(* IEC 61131-3 sources: ev-charging-controller/Communication, 3 files *)

(* ---- CanDecodeHelpers.st ---- *)
(* @brief Raw CAN field -> strict enum conversions
 *
 *  Strict enums cannot be assigned from integers, so each 2-bit field
 *  is mapped explicitly. Unknown codes fall back to the safe value.
 *)
FUNCTION F_ToContactorState : E_ContactorState
VAR_INPUT
    raw : BYTE;       (* 2-bit field, already shifted to bits 1:0 *)
END_VAR
    CASE raw OF
        0: F_ToContactorState := E_ContactorState.CTR_OPEN;
        1: F_ToContactorState := E_ContactorState.CTR_CLOSING;
        2: F_ToContactorState := E_ContactorState.CTR_CLOSED;
    ELSE
        F_ToContactorState := E_ContactorState.CTR_WELDED;
    END_CASE
END_FUNCTION

FUNCTION F_ToChargeProtocol : E_ChargeProtocol
VAR_INPUT
    raw : BYTE;       (* 2-bit field, bits 1:0 *)
END_VAR
    CASE raw OF
        1: F_ToChargeProtocol := E_ChargeProtocol.PROTO_DIN70121;
        2: F_ToChargeProtocol := E_ChargeProtocol.PROTO_ISO15118;
    ELSE
        F_ToChargeProtocol := E_ChargeProtocol.PROTO_UNKNOWN;
    END_CASE
END_FUNCTION

(* ---- ChargerCAN_RX.st ---- *)
(* @brief CAN receive handler for BMS and EVSE messages
 *
 *  Decodes incoming CAN frames and populates:
 *    - g_bms.rx   (5 messages from BMS on CAN3)
 *    - g_evse.rx   (3 messages from EVSE on CAN4)
 *
 *  Runs as PROGRAM on CycleCharge task (10ms).
 *  All multi-byte signals are little-endian (Intel byte order).
 *  J1939 extended 29-bit CAN identifiers.
 *)
PROGRAM PRG_ChargerCAN_RX
VAR
    (* ── BMS receive instances (CAN3) ── *)
    rxBmsPackData   : CanRx;
    rxBmsCellVolts  : CanRx;
    rxBmsCellTemps  : CanRx;
    rxBmsCtrStatus  : CanRx;
    rxBmsLimits     : CanRx;

    (* ── EVSE receive instances (CAN4) ── *)
    rxEvseStatus    : CanRx;
    rxEvseMetering  : CanRx;
    rxEvseProtocol  : CanRx;

    (* ── Data buffers ── *)
    dataBmsPackData   : ARRAY[0..7] OF BYTE;
    dataBmsCellVolts  : ARRAY[0..7] OF BYTE;
    dataBmsCellTemps  : ARRAY[0..7] OF BYTE;
    dataBmsCtrStatus  : ARRAY[0..7] OF BYTE;
    dataBmsLimits     : ARRAY[0..7] OF BYTE;
    dataEvseStatus    : ARRAY[0..7] OF BYTE;
    dataEvseMetering  : ARRAY[0..7] OF BYTE;
    dataEvseProtocol  : ARRAY[0..7] OF BYTE;

    (* ── Decode helpers ── *)
    rawU16 : UINT;
END_VAR

(* ══════════════════════════════════════════════════════════════
   CAN3 — BMS MESSAGES (5 receive)
   ══════════════════════════════════════════════════════════════ *)

(* ── 1. BMS Pack Data ── *)
rxBmsPackData(
    iCAN           := ADR(g_can3),
    iCanId         := CAN_ID_BMS_PACK_DATA,
    iCanIdExtended := TRUE,
    iTimeoutLimit  := T#500MS,
    oData          => dataBmsPackData
);
IF rxBmsPackData.oNewData THEN
    (* Pack voltage: bytes 0-1, 0.1 V/bit, little-endian *)
    rawU16 := BYTE_TO_UINT(dataBmsPackData[0])
           OR SHL(BYTE_TO_UINT(dataBmsPackData[1]), 8);
    g_bms.rx.packVoltage := UINT_TO_REAL(rawU16) * 0.1;

    (* Pack current: bytes 2-3, 0.1 A/bit, offset -3200 A *)
    rawU16 := BYTE_TO_UINT(dataBmsPackData[2])
           OR SHL(BYTE_TO_UINT(dataBmsPackData[3]), 8);
    g_bms.rx.packCurrent := (UINT_TO_REAL(rawU16) * 0.1) - 3200.0;

    (* SOC: byte 4, 1 %/bit *)
    g_bms.rx.soc := dataBmsPackData[4];

    (* SOH: byte 5, 1 %/bit *)
    g_bms.rx.soh := dataBmsPackData[5];

    g_bms.commOk     := TRUE;
    g_bms.lastRxTime := g_vcu.systemTime;
END_IF

(* ── 2. BMS Cell Voltages ── *)
rxBmsCellVolts(
    iCAN           := ADR(g_can3),
    iCanId         := CAN_ID_BMS_CELL_VOLTS,
    iCanIdExtended := TRUE,
    iTimeoutLimit  := T#500MS,
    oData          => dataBmsCellVolts
);
IF rxBmsCellVolts.oNewData THEN
    (* Cell voltage min: bytes 0-1, 1 mV/bit *)
    g_bms.rx.cellVoltageMin :=
        BYTE_TO_UINT(dataBmsCellVolts[0])
        OR SHL(BYTE_TO_UINT(dataBmsCellVolts[1]), 8);

    (* Cell voltage max: bytes 2-3, 1 mV/bit *)
    g_bms.rx.cellVoltageMax :=
        BYTE_TO_UINT(dataBmsCellVolts[2])
        OR SHL(BYTE_TO_UINT(dataBmsCellVolts[3]), 8);

    g_bms.commOk     := TRUE;
    g_bms.lastRxTime := g_vcu.systemTime;
END_IF

(* ── 3. BMS Cell Temperatures ── *)
rxBmsCellTemps(
    iCAN           := ADR(g_can3),
    iCanId         := CAN_ID_BMS_CELL_TEMPS,
    iCanIdExtended := TRUE,
    iTimeoutLimit  := T#500MS,
    oData          => dataBmsCellTemps
);
IF rxBmsCellTemps.oNewData THEN
    (* All temps: 1 C/bit, offset -40 C *)
    g_bms.rx.cellTempMin := BYTE_TO_INT(dataBmsCellTemps[0]) - 40;
    g_bms.rx.cellTempMax := BYTE_TO_INT(dataBmsCellTemps[1]) - 40;
    g_bms.rx.inletTemp   := BYTE_TO_INT(dataBmsCellTemps[2]) - 40;
    g_bms.rx.cableTemp   := BYTE_TO_INT(dataBmsCellTemps[3]) - 40;
    g_bms.rx.coolantTemp := BYTE_TO_INT(dataBmsCellTemps[4]) - 40;

    g_bms.commOk     := TRUE;
    g_bms.lastRxTime := g_vcu.systemTime;
END_IF

(* ── 4. BMS Contactor Status ── *)
rxBmsCtrStatus(
    iCAN           := ADR(g_can3),
    iCanId         := CAN_ID_BMS_CTR_STATUS,
    iCanIdExtended := TRUE,
    iTimeoutLimit  := T#500MS,
    oData          => dataBmsCtrStatus
);
IF rxBmsCtrStatus.oNewData THEN
    (* Byte 0: four 2-bit contactor feedback fields *)
    g_bms.rx.fbkMainPos   := F_ToContactorState(dataBmsCtrStatus[0] AND BYTE#16#03);
    g_bms.rx.fbkMainNeg   := F_ToContactorState(SHR(dataBmsCtrStatus[0] AND BYTE#16#0C, 2));
    g_bms.rx.fbkPrecharge := F_ToContactorState(SHR(dataBmsCtrStatus[0] AND BYTE#16#30, 4));
    g_bms.rx.fbkAcLine    := F_ToContactorState(SHR(dataBmsCtrStatus[0] AND BYTE#16#C0, 6));

    (* Byte 1: summary flags *)
    g_bms.rx.contactorClosed := (dataBmsCtrStatus[1] AND 16#01) <> 0;
    (* Weld is a latched fault: the BMS can set it, never clear it *)
    IF (dataBmsCtrStatus[1] AND 16#02) <> 0 THEN
        g_bms.rx.weldDetected := TRUE;
    END_IF

    g_bms.commOk     := TRUE;
    g_bms.lastRxTime := g_vcu.systemTime;
END_IF

(* ── 5. BMS Limits ── *)
rxBmsLimits(
    iCAN           := ADR(g_can3),
    iCanId         := CAN_ID_BMS_LIMITS,
    iCanIdExtended := TRUE,
    iTimeoutLimit  := T#500MS,
    oData          => dataBmsLimits
);
IF rxBmsLimits.oNewData THEN
    (* Max charge current: bytes 0-1, 0.1 A/bit *)
    rawU16 := BYTE_TO_UINT(dataBmsLimits[0])
           OR SHL(BYTE_TO_UINT(dataBmsLimits[1]), 8);
    g_bms.rx.maxChargeCurrent := UINT_TO_REAL(rawU16) * 0.1;

    (* Max discharge current: bytes 2-3, 0.1 A/bit *)
    rawU16 := BYTE_TO_UINT(dataBmsLimits[2])
           OR SHL(BYTE_TO_UINT(dataBmsLimits[3]), 8);
    g_bms.rx.maxDischargeCurrent := UINT_TO_REAL(rawU16) * 0.1;

    g_bms.commOk     := TRUE;
    g_bms.lastRxTime := g_vcu.systemTime;
END_IF

END_PROGRAM

(* ---- ChargerCAN_TX.st ---- *)
(* @brief CAN transmit handler for BMS and EVSE messages
 *
 *  Encodes outgoing CAN frames from:
 *    - g_bms.tx    (2 messages to BMS on CAN3)
 *    - g_evse.tx   (3 messages to EVSE on CAN4)
 *
 *  Runs as PROGRAM on CycleCharge task (10ms).
 *  All multi-byte signals are little-endian (Intel byte order).
 *  J1939 extended 29-bit CAN identifiers.
 *
 *  Transmit rates:
 *    50ms  — BMS Charge Cmd   (safety-critical contactor commands)
 *    100ms — Charge Request, Charge Params, BMS Charge Lim
 *    250ms — Charge Status    (informational)
 *)
PROGRAM PRG_ChargerCAN_TX
VAR
    (* ── EVSE transmit instances (CAN4) ── *)
    txChargeRequest : CanTx;
    txChargeParams  : CanTx;
    txChargeStatus  : CanTx;

    (* ── BMS transmit instances (CAN3) ── *)
    txBmsChargeCmd  : CanTx;
    txBmsChargeLim  : CanTx;

    (* ── Data buffers ── *)
    dataChargeRequest : ARRAY[0..7] OF BYTE;
    dataChargeParams  : ARRAY[0..7] OF BYTE;
    dataChargeStatus  : ARRAY[0..7] OF BYTE;
    dataBmsChargeCmd  : ARRAY[0..7] OF BYTE;
    dataBmsChargeLim  : ARRAY[0..7] OF BYTE;

    (* ── Encode helpers ── *)
    encU16 : UINT;
END_VAR

(* ══════════════════════════════════════════════════════════════
   CAN4 — EVSE MESSAGES (3 transmit)
   ══════════════════════════════════════════════════════════════ *)

(* ── 9. Charge Request  (100ms) ── *)

(* Byte 0: state [3:0] + mode [5:4] *)
dataChargeRequest[0] := TO_BYTE(g_evse.tx.state) AND 16#0F;
dataChargeRequest[0] := dataChargeRequest[0]
    OR SHL(TO_BYTE(g_evse.tx.mode) AND BYTE#16#03, 4);

(* Byte 1: alive counter *)
IF g_evse.tx.aliveCounter < ALIVE_COUNTER_MAX THEN
    g_evse.tx.aliveCounter := g_evse.tx.aliveCounter + 1;
ELSE
    g_evse.tx.aliveCounter := 0;
END_IF
dataChargeRequest[1] := g_evse.tx.aliveCounter;

(* Byte 2: chargeEnable [bit 0] + emergencyStop [bit 1] *)
dataChargeRequest[2] := 0;
IF g_evse.tx.chargeEnable THEN
    dataChargeRequest[2] := dataChargeRequest[2] OR 16#01;
END_IF
IF g_evse.tx.emergencyStop THEN
    dataChargeRequest[2] := dataChargeRequest[2] OR 16#02;
END_IF

(* Bytes 3-7: reserved *)
dataChargeRequest[3] := 0;
dataChargeRequest[4] := 0;
dataChargeRequest[5] := 0;
dataChargeRequest[6] := 0;
dataChargeRequest[7] := 0;

txChargeRequest(
    iEnable        := TRUE,
    iCAN           := ADR(g_can4),
    iForceSend     := FALSE,
    iTransmitRate  := T#100MS,
    iCanId         := CAN_ID_CHARGE_REQUEST,
    iCanIdExtended := TRUE,
    iByteCount     := 8,
    iData          := dataChargeRequest
);

(* ── 10. Charge Params  (100ms) ── *)

(* Bytes 0-1: target voltage, 0.1 V/bit, little-endian *)
encU16 := REAL_TO_UINT(g_evse.tx.targetVoltage * 10.0);
dataChargeParams[0] := TO_BYTE(encU16 AND 16#FF);
dataChargeParams[1] := TO_BYTE(SHR(encU16, 8) AND 16#FF);

(* Bytes 2-3: target current, 0.1 A/bit, little-endian *)
encU16 := REAL_TO_UINT(g_evse.tx.targetCurrent * 10.0);
dataChargeParams[2] := TO_BYTE(encU16 AND 16#FF);
dataChargeParams[3] := TO_BYTE(SHR(encU16, 8) AND 16#FF);

(* Byte 4: CC/CV flag *)
dataChargeParams[4] := g_evse.tx.ccCvFlag;

(* Byte 5: battery SOC *)
dataChargeParams[5] := g_evse.tx.soc;

(* Bytes 6-7: reserved *)
dataChargeParams[6] := 0;
dataChargeParams[7] := 0;

txChargeParams(
    iEnable        := TRUE,
    iCAN           := ADR(g_can4),
    iForceSend     := FALSE,
    iTransmitRate  := T#100MS,
    iCanId         := CAN_ID_CHARGE_PARAMS,
    iCanIdExtended := TRUE,
    iByteCount     := 8,
    iData          := dataChargeParams
);

(* ── 11. Charge Status  (250ms) ── *)

(* Byte 0: vehicle state *)
dataChargeStatus[0] := TO_BYTE(g_evse.tx.vehicleState);

(* Byte 1: precharge step *)
dataChargeStatus[1] := TO_BYTE(g_evse.tx.prechargeStep);

(* Byte 2: parkingBrake [bit 0] + ignitionOn [bit 1] + chargeComplete [bit 2] *)
dataChargeStatus[2] := 0;
IF g_evse.tx.parkingBrake THEN
    dataChargeStatus[2] := dataChargeStatus[2] OR 16#01;
END_IF
IF g_evse.tx.ignitionOn THEN
    dataChargeStatus[2] := dataChargeStatus[2] OR 16#02;
END_IF
IF g_evse.tx.chargeComplete THEN
    dataChargeStatus[2] := dataChargeStatus[2] OR 16#04;
END_IF

(* Bytes 3-7: reserved *)
dataChargeStatus[3] := 0;
dataChargeStatus[4] := 0;
dataChargeStatus[5] := 0;
dataChargeStatus[6] := 0;
dataChargeStatus[7] := 0;

txChargeStatus(
    iEnable        := TRUE,
    iCAN           := ADR(g_can4),
    iForceSend     := FALSE,
    iTransmitRate  := T#250MS,
    iCanId         := CAN_ID_CHARGE_STATUS,
    iCanIdExtended := TRUE,
    iByteCount     := 8,
    iData          := dataChargeStatus
);

(* ══════════════════════════════════════════════════════════════
   CAN3 — BMS MESSAGES (2 transmit)
   ══════════════════════════════════════════════════════════════ *)

(* ── 12. BMS Charge Command  (50ms — safety critical) ── *)

(* Byte 0: contactor commands as bit flags *)
dataBmsChargeCmd[0] := 0;
IF g_bms.tx.cmdMainPos THEN
    dataBmsChargeCmd[0] := dataBmsChargeCmd[0] OR 16#01;
END_IF
IF g_bms.tx.cmdMainNeg THEN
    dataBmsChargeCmd[0] := dataBmsChargeCmd[0] OR 16#02;
END_IF
IF g_bms.tx.cmdPrecharge THEN
    dataBmsChargeCmd[0] := dataBmsChargeCmd[0] OR 16#04;
END_IF
IF g_bms.tx.cmdAcLine THEN
    dataBmsChargeCmd[0] := dataBmsChargeCmd[0] OR 16#08;
END_IF

(* Byte 1: charge enable *)
IF g_bms.tx.chargeEnable THEN
    dataBmsChargeCmd[1] := 16#01;
ELSE
    dataBmsChargeCmd[1] := 16#00;
END_IF

(* Byte 2: charge mode *)
dataBmsChargeCmd[2] := TO_BYTE(g_bms.tx.chargeMode);

(* Bytes 3-7: reserved *)
dataBmsChargeCmd[3] := 0;
dataBmsChargeCmd[4] := 0;
dataBmsChargeCmd[5] := 0;
dataBmsChargeCmd[6] := 0;
dataBmsChargeCmd[7] := 0;

txBmsChargeCmd(
    iEnable        := TRUE,
    iCAN           := ADR(g_can3),
    iForceSend     := FALSE,
    iTransmitRate  := T#50MS,
    iCanId         := CAN_ID_BMS_CHARGE_CMD,
    iCanIdExtended := TRUE,
    iByteCount     := 8,
    iData          := dataBmsChargeCmd
);

(* ── 13. BMS Charge Limits  (100ms) ── *)

(* Bytes 0-1: target voltage, 0.1 V/bit, little-endian *)
encU16 := REAL_TO_UINT(g_bms.tx.targetVoltage * 10.0);
dataBmsChargeLim[0] := TO_BYTE(encU16 AND 16#FF);
dataBmsChargeLim[1] := TO_BYTE(SHR(encU16, 8) AND 16#FF);

(* Bytes 2-3: target current, 0.1 A/bit, little-endian *)
encU16 := REAL_TO_UINT(g_bms.tx.targetCurrent * 10.0);
dataBmsChargeLim[2] := TO_BYTE(encU16 AND 16#FF);
dataBmsChargeLim[3] := TO_BYTE(SHR(encU16, 8) AND 16#FF);

(* Byte 4: thermal derate factor, 1 %/bit *)
dataBmsChargeLim[4] := g_bms.tx.derateFactor;

(* Bytes 5-7: reserved *)
dataBmsChargeLim[5] := 0;
dataBmsChargeLim[6] := 0;
dataBmsChargeLim[7] := 0;

txBmsChargeLim(
    iEnable        := TRUE,
    iCAN           := ADR(g_can3),
    iForceSend     := FALSE,
    iTransmitRate  := T#100MS,
    iCanId         := CAN_ID_BMS_CHARGE_LIM,
    iCanIdExtended := TRUE,
    iByteCount     := 8,
    iData          := dataBmsChargeLim
);

END_PROGRAM
